TYPE DigitalOutputBase_1FE0D5EE :
STRUCT
END_STRUCT
END_TYPE

(* stored: Version 1.1.0.1, ProductVersion 3.1.4024.9
   DUT DigitalOutputBase_1FE0D5EE: Id {9b44b319-ab2b-016f-2b33-7e788ac6bd90} *)
